// TIA Portal V18 export
TYPE "AO"
// stored: IsFailsafeCompliant false
   STRUCT
      VFD : Int;
      "SPARE AO" : Int;
   END_STRUCT;
END_TYPE
